TYPE TcoCvirII_Config :
STRUCT
	
END_STRUCT
END_TYPE

(* stored: Version 1.1.0.1
   DUT TcoCvirII_Config: Id {4a6a36dc-b4de-4546-9e5f-cdeae6eb67ea} *)
